# EPICS alarm handler configuration: mps_database/bare/alarms/areas/mpln_ltuh_mp04.alhConfig
GROUP NULL MPLN:LTUH:MP04:1
$ALIAS MPS Link Node 133
$GUIDANCE
LTUH MPS
   Group Name: MPLN:LTUH:MP04:1
   Summary PV:  MPLN:LTUH:MP04:1:STATSUMY
$END
CHANNEL  MPLN:LTUH:MP04:1    MPLN:LTUH:MP04:1:MPS_EN_RBV		-----
CHANNEL  MPLN:LTUH:MP04:1    MPLN:LTUH:MP04:1:LC1_MODE_RBV		-----
